      # calculate rxryrz
      # rotate 180 degrees about x. then rotate (90 deg + heading3 degrees) about z ccw
      m1 = get_rotation_matrix_from_description("x", -1, 180 * pi / 180)
      m2 = get_rotation_matrix_from_description("z", 1, heading3 + pi/2)
      m3 = multiply_matrix(m2, m1) #we rotate m1 first then m2, so we multiply in backwards order: 2 then 1
      rxryrz = convert_matrix_to_axang(m3)
      rx = rxryrz[0]
      ry = rxryrz[1]
      rz = rxryrz[2]
      point201 = p[p201x, p201y, z, rx, ry, rz]

      # calculate point 201's preheat
      pushtipforward2 = 0.012 - pushtipforward # 12 mm forward to clear the existing extrudant (but still have the extrudant from this extrusion join the existing). subtract from previous to make it constant even if you change pushtipforward1
      preheatdistance = 0.010 # 10 mm . above what it would be pushed down
      point201a = p[p201x, p201y, z + preheatdistance, rx, ry, rz]
      p201bx = p201x + l2delxunit * pushtipforward2
      p201by = p201y + l2delyunit * pushtipforward2
      point201b = p[p201bx, p201by, z + preheatdistance, rx, ry, rz]
      point201c = p[p201bx, p201by, z, rx, ry, rz]

      # calculate point 202
      p202x = p201x + wd3 * l2delxunit
      p202y = p201y + wd3 * l2delyunit
      point202 = p[p202x, p202y, z, rx, ry, rz]

      struct2 = struct(point1=point1, point2=point2, point3=point3, point4=point4, point5=point5, point201=point201, point202=point202, point201a=point201a, point201b=point201b, point201c=point201c, point2a=point2a)
      return struct2
  end

  def calculate_AtS_points_cover_right(struct1, leftwallthick, rightwallthick):
      # get the stuff from the struct
      pointintersect = struct1[0]
      heading1 = struct1[1]
      heading2 = struct1[2]
      heading3 = struct1[3]
      l1delxunit = struct1[4]
      l1delyunit = struct1[5]
      l2delxunit = struct1[6]
      l2delyunit = struct1[7]

      # FIND THE POINTS ON THE LINES OF THE FIRST TURN PATH
      # find locations 8 inches away from  intersect point
      # CONST
      welddistance1 = 6 # first path first leg (down)
      welddistance2 = 4 # first path second leg (under) # inches
      welddistance3 = 6 # second path (back away) # inches

      wd1 = welddistance1 * 25.4 / 1000
      wd2 = welddistance2 * 25.4 / 1000
      wd3 = welddistance3 * 25.4 / 1000
      leftwallthickmm = leftwallthick * 25.4 / 1000 # in this step corner right, this is distance from left edge
      rightwallthickmm =  rightwallthick * 25.4 / 1000 # in this step corner right, this is distance from right edge

      # first, check if we need a lift column raise
      # (we do, because for maximum reach we want to make the lift pedestal be even with the top of the covers)
      zpi = pointintersect[2]
      if zpi > 0:
          liftcolumnzneeded = zpi * 1000.0 # the robot uses coordinates in meters, but the lift column uses coordinates in mm
          z = 0
      else:
          z = zpi
      end

      # first, calculate the location of the top of the vertical chamfer (where point2 would be if there weren't any circle motion)
      x = pointintersect[0] + l1delxunit * leftwallthickmm
      y = pointintersect[1] + l1delyunit * leftwallthickmm
      #z = pointintersect[2] # replaced by z of lift column (directly above)
      pointtopvcham = p[x, y, z, 0, 0, 0]

      # calculate the rxryrz for the gun when it's at point1
      # start with rxryrz = 0,0,0 (gun facing up, preheat facing y+ axis.
      # rotate it 180 degrees about x axis. gun facing down, preheat facing y- axis
      # rotate it about 135 degrees ccw about z axis. x+ to heading3 is about 225 degrees. so our angle is heading3 - 90 degrees
      m1 = get_rotation_matrix_from_description("x", -1, 180 * pi / 180) # rotation 1: 180 degrees forward about x axis
      m2 = get_rotation_matrix_from_description("z", 1, heading3 - pi/2) # rotation 2
      m3 = multiply_matrix(m2, m1) #we rotate m1 first then m2, so we multiply in backwards order: 2 then 1
      rxryrz = convert_matrix_to_axang(m3)
      rx = rxryrz[0]
      ry = rxryrz[1]
      rz = rxryrz[2]

      # next, calculate point1
      p1x = x + l2delxunit * wd1
      p1y = y + l2delyunit * wd1
      point1 = p[p1x, p1y, z, rx, ry, rz]

      # the round over distance is the distance from pointbottomvcham to point2 (which will be the same as distance to p4)
      roundoverdistance = 0.05
      rod = roundoverdistance * 25.4 / 1000
      p2x = x + l2delxunit * rod
      p2y = y + l2delyunit * rod
      point2 = p[p2x, p2y, z, rx, ry, rz]

      # make point2a, colinear between p1 and p2, which will be the place the welder shuts off during motion
      wtod = 0.015 # weldturnoffdistance # meters from pointtopvcham # 10 mm (1.0 seconds)
      p2ax = x + l2delxunit * wtod
      p2ay = y + l2delyunit * wtod
      point2a = p[p2ax, p2ay, z, rx, ry, rz]

      # calculate the rxryrz for facing the down the right side of the box
      # rotate about x 90 (forward). then rotate about z ~ 135 (ccw)
      m1 = get_rotation_matrix_from_description("x", -1, 90 * pi / 180)
      m2 = get_rotation_matrix_from_description("z", 1, heading3 - pi/2)
      m3 = multiply_matrix(m2, m1) #we rotate m1 first then m2, so we multiply in backwards order: 2 then 1
      rxryrz = convert_matrix_to_axang(m3)
      rx = rxryrz[0]
      ry = rxryrz[1]
      rz = rxryrz[2]

      # calculate point4
      point4 = p[x, y, z - rod, rx, ry, rz]

      # calculate point5
      point5 = p[x, y, z - wd2, rx, ry, rz]

      # calculate point3
      # we know that the angle is exactly 90 degrees
      delta = calc_rod_midpoint_90deg(rod)
      p3z = z - delta
      p3x = x + delta * l2delxunit
      p3y = y + delta * l2delyunit

      # calculate rxryrz
      m1 = get_rotation_matrix_from_description("x", -1, 135 * pi / 180) # rotation 1: 135 degrees forward about x axis
      m2 = get_rotation_matrix_from_description("z", 1, heading3 - pi/2)
      m3 = multiply_matrix(m2, m1) #we rotate m1 first then m2, so we multiply in backwards order: 2 then 1
      rxryrz = convert_matrix_to_axang(m3)
      rx = rxryrz[0]
      ry = rxryrz[1]
      rz = rxryrz[2]
      point3 = p[p3x, p3y, p3z, rx, ry, rz]

      #todo: calculate trail out point

      # calculate back-away (points 201 and 202)
      pushtipforward = 0.006 # 6 millimeters forward. the tip needs to clear the capping wall's angled chamfer to not BONK when getting into position
      p201x = x + l2delxunit * rightwallthickmm + l1delxunit * pushtipforward
      p201y = y + l2delyunit * rightwallthickmm + l1delyunit * pushtipforward

      # calculate rxryrz
      # rotate 180 degrees about x. then rotate (90 deg + heading1 degrees) about z ccw
      m1 = get_rotation_matrix_from_description("x", -1, 180 * pi / 180)
      m2 = get_rotation_matrix_from_description("z", 1, heading1 + pi/2)
      m3 = multiply_matrix(m2, m1) #we rotate m1 first then m2, so we multiply in backwards order: 2 then 1
      rxryrz = convert_matrix_to_axang(m3)
      rx = rxryrz[0]
      ry = rxryrz[1]
      rz = rxryrz[2]
      point201 = p[p201x, p201y, z, rx, ry, rz]

      # calculate point 201's preheat
      pushtipforward2 = 0.012 - pushtipforward # 12 mm forward to clear the existing extrudant (but still have the extrudant from this extrusion join the existing). subtract from previous to make it constant even if you change pushtipforward1
      preheatdistance = 0.010 # 10 mm . above what it would be pushed down
      point201a = p[p201x, p201y, z + preheatdistance, rx, ry, rz]
      p201bx = p201x + l1delxunit * pushtipforward2
      p201by = p201y + l1delyunit * pushtipforward2
      point201b = p[p201bx, p201by, z + preheatdistance, rx, ry, rz]
      point201c = p[p201bx, p201by, z, rx, ry, rz]

      # calculate point 202
      p202x = p201x + wd3 * l1delxunit
      p202y = p201y + wd3 * l1delyunit
      point202 = p[p202x, p202y, z, rx, ry, rz]

      struct2 = struct(point1=point1, point2=point2, point3=point3, point4=point4, point5=point5, point201=point201, point202=point202, point201a=point201a, point201b=point201b, point201c=point201c, point2a=point2a)
      return struct2
  end
  $ 16 "path_pre≔get_corner_homing_45_pathpoints_cover(tp)"
  global path_pre=get_corner_homing_45_pathpoints_cover(tp)
  $ 17 "ph1≔path_pre[0]"
  global ph1=path_pre[0]
  $ 18 "ph2≔path_pre[1]"
  global ph2=path_pre[1]
  $ 19 "ph3≔path_pre[2]"
  global ph3=path_pre[2]
  $ 20 "ph4≔path_pre[3]"
  global ph4=path_pre[3]
  $ 21 "ph5≔path_pre[4]"
  global ph5=path_pre[4]
  $ 22 "ph6≔path_pre[5]"
  global ph6=path_pre[5]
  $ 23 "ph7≔path_pre[6]"
  global ph7=path_pre[6]
  $ 26 "MoveL"
  $ 27 "ph1" "breakAfter"
  movel(ph1, a=0.2, v=0.25)
  $ 28 "ph2" "breakAfter"
  movel(ph2, a=0.2, v=0.25)
  $ 29 "MoveL"
  $ 30 "Direction: Base"
  global move_thread_flag_30=0
  thread move_thread_30():
    enter_critical
    move_thread_flag_30 = 1
    local towardsPos=calculate_point_to_move_towards(p[0.0,0.0,0.0,0.0,0.0,0.0], [-1,-1.0,0.0], 1000.0)
    movel(towardsPos, a=0.1, v=0.02)
    move_thread_flag_30 = 2
    exit_critical
  end
  move_thread_flag_30 = 0
  move_thread_han_30 = run move_thread_30()
  while (True):
    local targetTcpDirection=get_target_tcp_speed()
    local stepsToRetract=tool_contact(direction=targetTcpDirection)
    if (stepsToRetract > 0):
      kill move_thread_han_30
      stopl(3.0)
      local backTrackMovement=get_actual_joint_positions_history(stepsToRetract)
      local contactPose=get_forward_kin(backTrackMovement)
      local posDir=[targetTcpDirection[0],targetTcpDirection[1],targetTcpDirection[2]]
      local retractTo=contactPose
      if (norm(posDir) > 1e-6):
        local normalizedPosDir=normalize(posDir)
        local additionalRetraction=p[normalizedPosDir[0] * 0.0, normalizedPosDir[1] * 0.0, normalizedPosDir[2] * 0.0, 0, 0, 0]
        retractTo = pose_sub(contactPose, additionalRetraction)
      end
      movel(retractTo, a=3.0, v=0.1)
      $ 31 "Until (tool_contact_detection)"
      break
    end
    sync()
  end
  $ 32 "p11≔get_actual_tcp_pose()"
  global p11= get_actual_tcp_pose ()
  $ 33 "MoveJ"
  $ 34 "ph2" "breakAfter"
  movej(ph2, a=1.3962634015954636, v=1.0471975511965976)
  $ 35 "ph3" "breakAfter"
  movej(ph3, a=1.3962634015954636, v=1.0471975511965976)
  $ 36 "MoveL"
  $ 37 "Direction: Base"
  global move_thread_flag_37=0
  thread move_thread_37():
    enter_critical
    move_thread_flag_37 = 1
    local towardsPos=calculate_point_to_move_towards(p[0.0,0.0,0.0,0.0,0.0,0.0], [-1,-1.0,0.0], 1000.0)
    movel(towardsPos, a=0.1, v=0.02)
    move_thread_flag_37 = 2
    exit_critical
  end
  move_thread_flag_37 = 0
  move_thread_han_37 = run move_thread_37()
  while (True):
    local targetTcpDirection=get_target_tcp_speed()
    local stepsToRetract=tool_contact(direction=targetTcpDirection)
    if (stepsToRetract > 0):
      kill move_thread_han_37
      stopl(3.0)
      local backTrackMovement=get_actual_joint_positions_history(stepsToRetract)
      local contactPose=get_forward_kin(backTrackMovement)
      local posDir=[targetTcpDirection[0],targetTcpDirection[1],targetTcpDirection[2]]
      local retractTo=contactPose
      if (norm(posDir) > 1e-6):
        local normalizedPosDir=normalize(posDir)
        local additionalRetraction=p[normalizedPosDir[0] * 0.0, normalizedPosDir[1] * 0.0, normalizedPosDir[2] * 0.0, 0, 0, 0]
        retractTo = pose_sub(contactPose, additionalRetraction)
      end
      movel(retractTo, a=3.0, v=0.1)
      $ 38 "Until (tool_contact_detection)"
      break
    end
    sync()
  end
  $ 46 "p12≔get_actual_tcp_pose()"
  global p12= get_actual_tcp_pose ()
  $ 47 "MoveJ"
  $ 48 "ph3" "breakAfter"
  movej(ph3, a=1.3962634015954636, v=1.0471975511965976)
  $ 49 "MoveJ"
  $ 50 "ph1" "breakAfter"
  movej(ph1, a=1.3962634015954636, v=1.0471975511965976)
  $ 51 "MoveJ"
  $ 52 "Waypoint_3" "breakAfter"
  movej(get_inverse_kin(Waypoint_3_p, qnear=Waypoint_3_q), a=1.3962634015954636, v=1.0471975511965976)
  $ 53 "Waypoint_6" "breakAfter"
  movej(get_inverse_kin(Waypoint_6_p, qnear=Waypoint_6_q), a=1.3962634015954636, v=1.0471975511965976)
  $ 59 "MoveJ"
  $ 60 "ph4" "breakAfter"
  movej(ph4, a=1.3962634015954636, v=1.0471975511965976)
  $ 61 "MoveL"
  $ 62 "Direction: Base"
  global move_thread_flag_62=0
  thread move_thread_62():
    enter_critical
    move_thread_flag_62 = 1
    local towardsPos=calculate_point_to_move_towards(p[0.0,0.0,0.0,0.0,0.0,0.0], [-1.0,1.0,0.0], 1000.0)
    movel(towardsPos, a=0.1, v=0.02)
    move_thread_flag_62 = 2
    exit_critical
  end
  move_thread_flag_62 = 0
  move_thread_han_62 = run move_thread_62()
  while (True):
    local targetTcpDirection=get_target_tcp_speed()
    local stepsToRetract=tool_contact(direction=targetTcpDirection)
    if (stepsToRetract > 0):
      kill move_thread_han_62
      stopl(3.0)
      local backTrackMovement=get_actual_joint_positions_history(stepsToRetract)
      local contactPose=get_forward_kin(backTrackMovement)
      local posDir=[targetTcpDirection[0],targetTcpDirection[1],targetTcpDirection[2]]
      local retractTo=contactPose
      if (norm(posDir) > 1e-6):
        local normalizedPosDir=normalize(posDir)
        local additionalRetraction=p[normalizedPosDir[0] * 0.0, normalizedPosDir[1] * 0.0, normalizedPosDir[2] * 0.0, 0, 0, 0]
        retractTo = pose_sub(contactPose, additionalRetraction)
      end
      movel(retractTo, a=3.0, v=0.1)
      $ 63 "Until (tool_contact_detection)"
      break
    end
    sync()
  end
  $ 64 "p21≔get_actual_tcp_pose()"
  global p21= get_actual_tcp_pose ()
  $ 65 "MoveL"
  $ 66 "ph4" "breakAfter"
  movel(ph4, a=1.2, v=0.25)
  $ 69 "MoveJ"
  $ 71 "Waypoint_9" "breakAfter"
  movej(get_inverse_kin(Waypoint_9_p, qnear=Waypoint_9_q), a=1.3962634015954636, v=1.0471975511965976)
  $ 72 "MoveJ"
  $ 73 "Waypoint_16" "breakAfter"
  movej(get_inverse_kin(Waypoint_16_p, qnear=Waypoint_16_q), a=1.3962634015954636, v=1.0471975511965976)
  $ 74 "MoveJ"
  $ 75 "Waypoint_15" "breakAfter"
  movej(get_inverse_kin(Waypoint_15_p, qnear=Waypoint_15_q), a=1.3962634015954636, v=1.0471975511965976)
  $ 77 "MoveJ"
  $ 78 "ph6" "breakAfter"
  movej(ph6, a=1.3962634015954636, v=1.0471975511965976)
  $ 79 "MoveL"
  $ 80 "ph7" "breakAfter"
  movel(ph7, a=1.2, v=0.25)
  $ 81 "MoveL"
  $ 82 "Direction: Base Z-"
  global move_thread_flag_82=0
  thread move_thread_82():
    enter_critical
    move_thread_flag_82 = 1
    local towardsPos=calculate_point_to_move_towards(p[0.0,0.0,0.0,0.0,0.0,0.0], [0.0,0.0,-1.0], 1000.0)
    movel(towardsPos, a=0.1, v=0.02)
    move_thread_flag_82 = 2
    exit_critical
  end
  move_thread_flag_82 = 0
  move_thread_han_82 = run move_thread_82()
  while (True):
    local targetTcpDirection=get_target_tcp_speed()
    local stepsToRetract=tool_contact(direction=targetTcpDirection)
    if (stepsToRetract > 0):
      kill move_thread_han_82
      stopl(3.0)
      local backTrackMovement=get_actual_joint_positions_history(stepsToRetract)
      local contactPose=get_forward_kin(backTrackMovement)
      local posDir=[targetTcpDirection[0],targetTcpDirection[1],targetTcpDirection[2]]
      local retractTo=contactPose
      if (norm(posDir) > 1e-6):
        local normalizedPosDir=normalize(posDir)
        local additionalRetraction=p[normalizedPosDir[0] * 0.0, normalizedPosDir[1] * 0.0, normalizedPosDir[2] * 0.0, 0, 0, 0]
        retractTo = pose_sub(contactPose, additionalRetraction)
      end
      movel(retractTo, a=3.0, v=0.1)
      $ 83 "Until (tool_contact_detection)"
      break
    end
    sync()
  end
  $ 84 "p3≔get_actual_tcp_pose()"
  global p3= get_actual_tcp_pose ()
  $ 85 "MoveL"
  $ 86 "ph7" "breakAfter"
  movel(ph7, a=1.2, v=0.25)
  $ 87 "ph6" "breakAfter"
  movel(ph6, a=1.2, v=0.25)
  $ 88 "MoveJ"
  $ 89 "Waypoint_15" "breakAfter"
  movej(get_inverse_kin(Waypoint_15_p, qnear=Waypoint_15_q), a=1.3962634015954636, v=1.0471975511965976)
  $ 97 "Home"
  movej([-3.266929759358355, -1.2139462677784536, 1.5878387874396154, 1.1069165929565088, -0.0023738326664366483, -1.7891447305770605], a=1.3962634015954636, v=1.0471975511965976)
end
